(* PLC project Sem nome, Desconhecido Sem nome 1 *)
(* stored: creationDateTime 2023-08-18T11:33:02, modificationDateTime 2024-04-17T14:44:26 *)

PROGRAM program0
  VAR
    mqtt_connected : BOOL;
    MQTT_SEND1 : MQTT_SEND;
    MQTT_CONNECT0 : MQTT_CONNECT;
    TON0 : TON;
  END_VAR
  VAR
    TURNON AT %IX1.0 : BOOL;
    TURNOFF AT %IX1.1 : BOOL;
    RESET AT %IX1.2 : BOOL;
    PARTSENSOR AT %IX0.0 : BOOL;
    INDUCTIVE AT %IX0.1 : BOOL;
    PHOTOELECTRIC AT %IX0.4 : BOOL;
    PASSING AT %IX0.5 : BOOL;
    CONVEYOR AT %QX0.0 : BOOL;
    ACTUATOR1 AT %QX0.1 : BOOL;
    ACTUATOR2 AT %QX0.2 : BOOL;
    BLOCK AT %QX0.3 : BOOL;
  END_VAR
  VAR
    MEMORY : BOOL;
    MEMORY1 : BOOL;
    MEMORY2 : BOOL;
    MEMORY3 : BOOL;
    SILVERMEMORY : BOOL;
    BLACKMEMORY : BOOL;
    REDMEMORY : BOOL;
    MQTT_SEND2 : MQTT_SEND;
    MQTT_SEND3 : MQTT_SEND;
    MQTT_SEND4 : MQTT_SEND;
    MQTT_SEND5 : MQTT_SEND;
    MQTT_SEND6 : MQTT_SEND;
    MQTT_SEND7 : MQTT_SEND;
    MQTT_SEND8 : MQTT_SEND;
  END_VAR

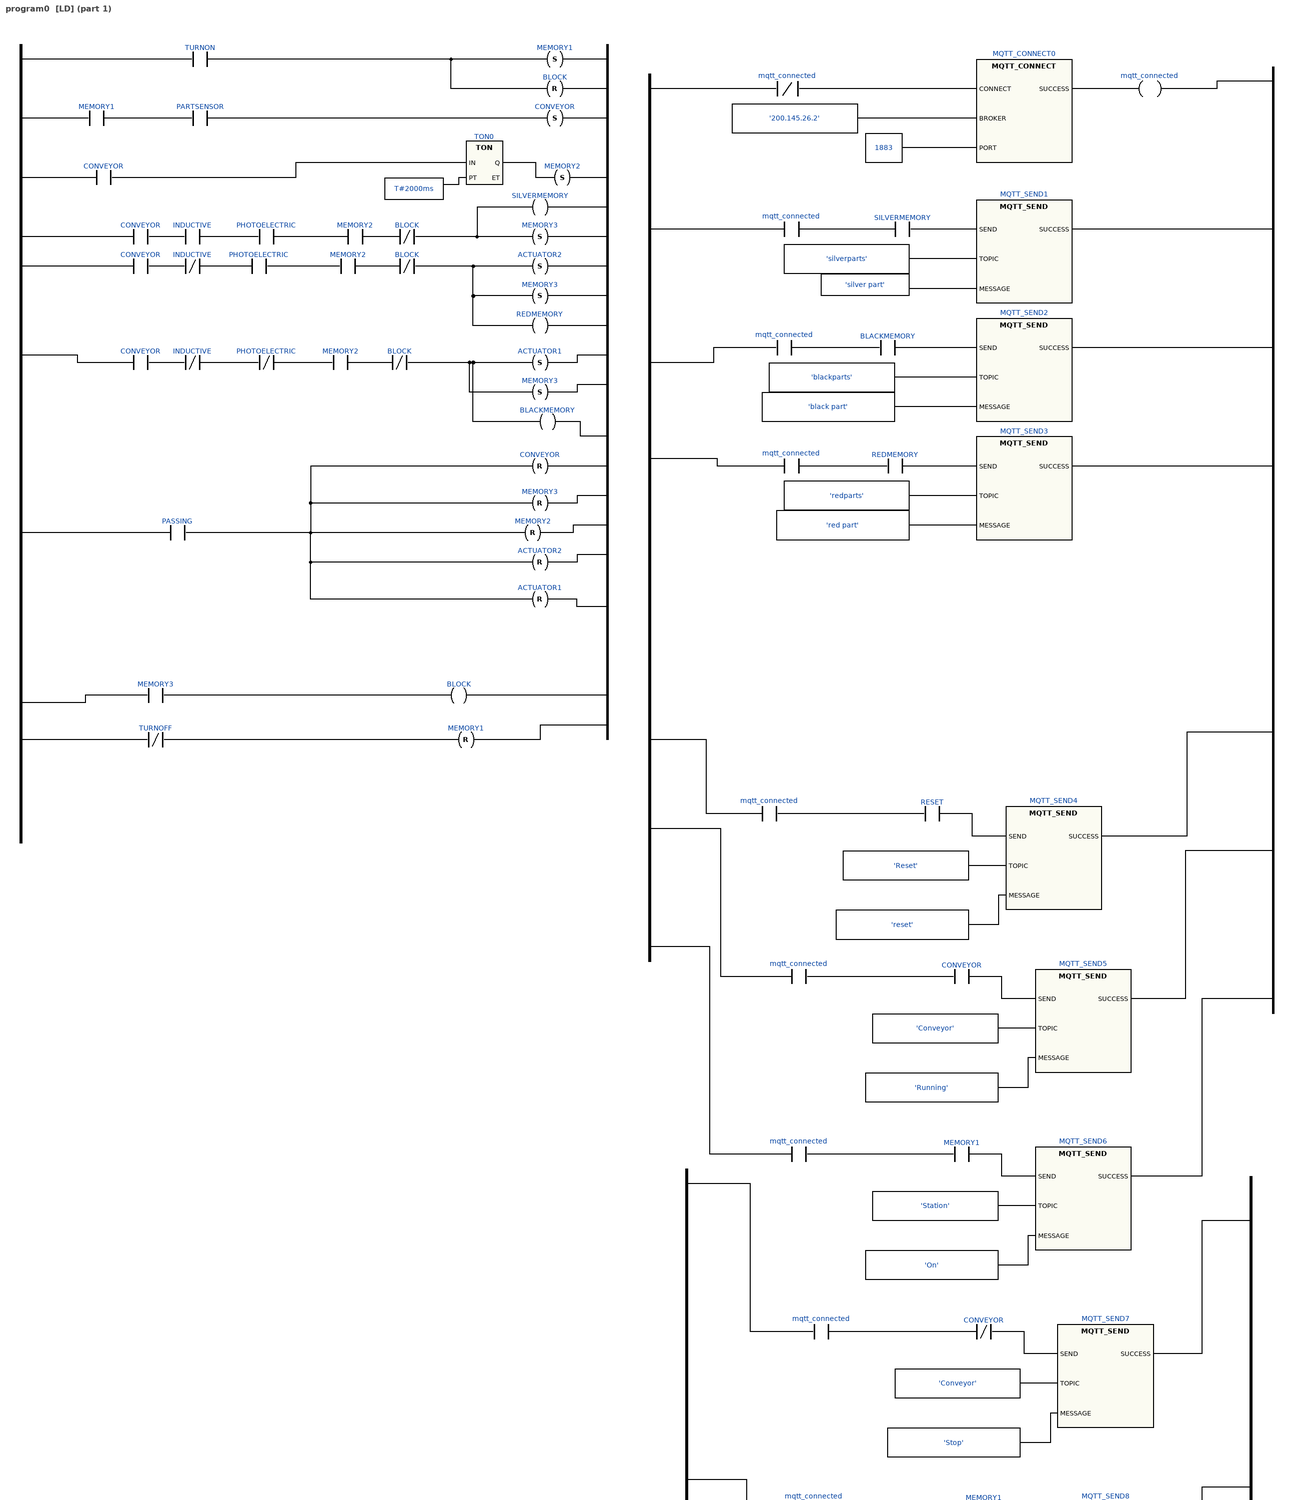
(* LD diagram, written out as Structured Text *)
MQTT_CONNECT0(CONNECT := NOT mqtt_connected, BROKER := '200.145.26.2', PORT := 1883);
mqtt_connected := MQTT_CONNECT0.SUCCESS;
IF CONVEYOR AND NOT INDUCTIVE AND NOT PHOTOELECTRIC AND MEMORY2 AND NOT BLOCK THEN MEMORY3 := TRUE; END_IF;
IF CONVEYOR AND NOT INDUCTIVE AND NOT PHOTOELECTRIC AND MEMORY2 AND NOT BLOCK THEN ACTUATOR1 := TRUE; END_IF;
IF CONVEYOR AND INDUCTIVE AND PHOTOELECTRIC AND MEMORY2 AND NOT BLOCK THEN MEMORY3 := TRUE; END_IF;
IF TURNON THEN MEMORY1 := TRUE; END_IF;
IF TURNON THEN BLOCK := FALSE; END_IF;
IF MEMORY1 AND PARTSENSOR THEN CONVEYOR := TRUE; END_IF;
IF CONVEYOR AND NOT INDUCTIVE AND PHOTOELECTRIC AND MEMORY2 AND NOT BLOCK THEN MEMORY3 := TRUE; END_IF;
IF CONVEYOR AND NOT INDUCTIVE AND PHOTOELECTRIC AND MEMORY2 AND NOT BLOCK THEN ACTUATOR2 := TRUE; END_IF;
TON0(IN := CONVEYOR, PT := T#2000ms);
IF TON0.Q THEN MEMORY2 := TRUE; END_IF;
IF PASSING THEN CONVEYOR := FALSE; END_IF;
IF PASSING THEN MEMORY3 := FALSE; END_IF;
IF PASSING THEN ACTUATOR1 := FALSE; END_IF;
IF PASSING THEN ACTUATOR2 := FALSE; END_IF;
IF PASSING THEN MEMORY2 := FALSE; END_IF;
BLOCK := MEMORY3;
IF NOT TURNOFF THEN MEMORY1 := FALSE; END_IF;
SILVERMEMORY := CONVEYOR AND INDUCTIVE AND PHOTOELECTRIC AND MEMORY2 AND NOT BLOCK;
REDMEMORY := CONVEYOR AND NOT INDUCTIVE AND PHOTOELECTRIC AND MEMORY2 AND NOT BLOCK;
BLACKMEMORY := CONVEYOR AND NOT INDUCTIVE AND NOT PHOTOELECTRIC AND MEMORY2 AND NOT BLOCK;
MQTT_SEND1(SEND := mqtt_connected AND SILVERMEMORY, TOPIC := 'silverparts', MESSAGE := 'silver part');
MQTT_SEND2(SEND := mqtt_connected AND BLACKMEMORY, TOPIC := 'blackparts', MESSAGE := 'black part');
MQTT_SEND3(SEND := mqtt_connected AND REDMEMORY, TOPIC := 'redparts', MESSAGE := 'red part');
MQTT_SEND4(SEND := mqtt_connected AND RESET, TOPIC := 'Reset', MESSAGE := 'reset');
MQTT_SEND5(SEND := mqtt_connected AND CONVEYOR, TOPIC := 'Conveyor', MESSAGE := 'Running');
MQTT_SEND6(SEND := mqtt_connected AND MEMORY1, TOPIC := 'Station', MESSAGE := 'On');
MQTT_SEND7(SEND := mqtt_connected AND NOT CONVEYOR, TOPIC := 'Conveyor', MESSAGE := 'Stop');
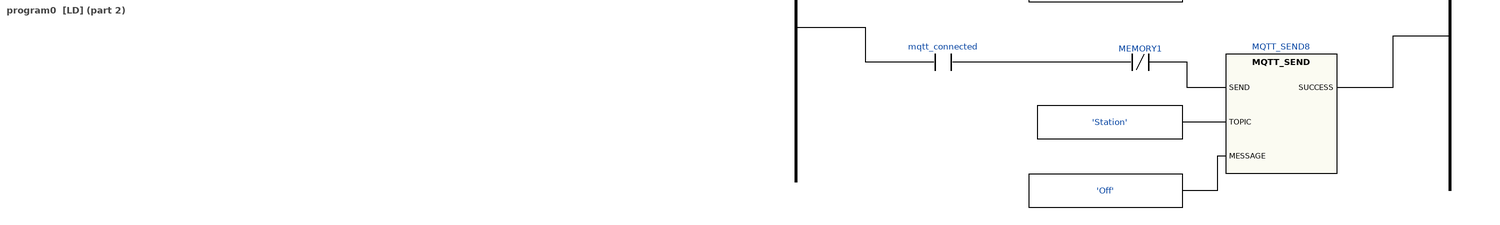
MQTT_SEND8(SEND := mqtt_connected AND NOT MEMORY1, TOPIC := 'Station', MESSAGE := 'Off');
END_PROGRAM

CONFIGURATION Config0
  RESOURCE Res0 ON PLC
    TASK task0(INTERVAL := T#20ms, PRIORITY := 0);
    PROGRAM instance0 WITH task0 : program0;
  END_RESOURCE
END_CONFIGURATION
